{attribute 'GeneratedUsingTerminal: EK1100-0000-0018'}
{attribute addProperty BoxType "EK1100-0000-0018"}
{attribute addProperty Id "Beckhoff_APS1xxxEK1122Beckhoff_APS1xxxEK1122_CD096C89258A_0002_APS1003_5000_0016APS1003_A49C5437320"}
{attribute addProperty CRC "3039580114"}
{attribute addProperty Size "578"}
TYPE Beckhoff_APS1xxx_B52C4FD2 EXTENDS EK1100_1FC0878B :
STRUCT
	{attribute addProperty Name "Beckhoff_APS1xxxEK1122"}
	{attribute addProperty PreviousPort "Beckhoff APS1xxx : B"}
	Beckhoff_APS1xxxEK1122 : Beckhoff_APS1xxxEK1122_CD096C89;
	{attribute addProperty Name "A_0002_APS1003_5000_0016"}
	{attribute addProperty PreviousPort "Beckhoff APS1xxxEK1122 : C"}
	A_0002_APS1003_5000_0016 : APS1003_A49C5437;
END_STRUCT
END_TYPE

(* stored: Version 1.2.0.0, ProductVersion 3.1.4024.9
   DUT Beckhoff_APS1xxx_B52C4FD2: Id {ea3798d4-fecb-4d1b-a7e2-fc901ec31477} *)
